(* Derived diagnostic status for an EtherCAT bridge terminal (EL6692/EL6695), which
links two independent EtherCAT masters (e.g. a subsystem PLC and an arbiter PLC).
LinkStatus gates DataStatus; ConnectionStatus is the two combined. *)
INTERFACE I_BridgeDiagnostics

(* Whether the bridge is established: local state, far device presence, far-side operational state. *)
PROPERTY LinkStatus : E_BridgeLinkStatus
GET
END_GET
END_PROPERTY

(* Combines WcState (whichever shape the box exposes) and the input toggle. *)
PROPERTY DataStatus : E_DataStatus
GET
END_GET
END_PROPERTY

(* Combined verdict: LinkStatus gates DataStatus. *)
PROPERTY ConnectionStatus : E_BridgeStatus
GET
END_GET
END_PROPERTY

END_INTERFACE

(* stored: Version 1.1.0.1
   Itf I_BridgeDiagnostics: Id {9d4e1a72-5b83-4c96-a017-6e2f8b3d5c04}
   Property LinkStatus: Id {b6f2c8a1-4d75-4e02-9a83-1c6f0e8b2d47}
   Get Get: Id {c1a4d0e6-2f83-4b57-8e0a-3d6c9f1b5a28}
   Property DataStatus: Id {e8b3f6c2-7a94-4d15-b028-4f7e2d9c6a53}
   Get Get: Id {f2c7d9e4-3b06-4a58-9c1d-5e8f3a0b6c74}
   Property ConnectionStatus: Id {a3d8e5f1-6c29-4b37-8d04-2f9c7e1a5b63}
   Get Get: Id {d4e9f0a2-7b31-4c48-9e15-3a0d8f2c6b74} *)
